FUNCTION_BLOCK FB_NormallyOpenPB IMPLEMENTS I_Pushbutton
VAR
	Input AT %I* : BOOL;
END_VAR

PROPERTY IsPressed : BOOL
GET
IsPressed := Input;
END_GET
END_PROPERTY

PROPERTY IsReleased : BOOL
GET
IsReleased := NOT Input;
END_GET
END_PROPERTY

END_FUNCTION_BLOCK

(* stored: Version 1.1.0.1, ProductVersion 3.1.4024.9
   POU FB_NormallyOpenPB: Id {206be575-3602-446b-bfbb-c57a428397fd}, SpecialFunc None
   Property IsPressed: Id {4f8940d5-542a-4841-91ec-44f7c53db87a}
   Get Get: Id {8f73b76e-b57f-4c34-87d3-87e7e2b903a2}
   Property IsReleased: Id {6cbd2a12-85f2-4fad-b2df-222bc8a1882d}
   Get Get: Id {a448a22e-897c-49bc-adc7-faa363001e4f} *)
